// TwinCAT 3 PLC project plc_simple_move
// ProgramVersion: 3.1.0.8
// libraries:
//   Tc2_MC2, * (Beckhoff Automation GmbH)
//   Tc2_Standard, * (Beckhoff Automation GmbH)
//   Tc2_System, * (Beckhoff Automation GmbH)
//   Tc3_Interfaces, * (Beckhoff Automation GmbH)
//   Tc3_Module, * (Beckhoff Automation GmbH)
// project tree:
//   / PlcTask.TcTTO
//   POUs/ MAIN.TcPOU
// real-time tasks:
//   TASK PlcTask: cycle T#10ms, priority 20, ADS port 350
// motion (NC):
//   TASK NC-Task 1 SAF: cycle T#2ms, priority 4, ADS port 501
//   TASK NC-Task 1 SVB: cycle T#10ms, priority 8, ADS port 511
//   AXIS Axis 1 (id 1)
//     OtherSettings: AllowMotionCmdToSlave=true
//     encoder EncType=19
//       EncPara: MaxCount=#xffffffff
//     drive DrvType=16
//       DrvPara: MaxCount=#xffffffff
//         TimeComp: TaskDelayCycles=1
//     controller CtrType=1
//       CtrPara: PriorControlFactor=1
//         Observer: BandWidth=20
// I/O:
//   DEVICE Device 5 (EtherCAT), AmsNetId 5.39.221.128.6.1
//     Drive 12 (Elmo Drive) [Gold EtherCAT GCON Drive Rev:0x000103F6]
// variable links:
//   NC-Task 1 SAF/Axes/Axis 1 <-> Device 5 (EtherCAT)/Drive 12 (Elmo Drive)
//     Drive/Inputs/In/nDcOutputTime <-> InfoData/DcOutputShift
//     Drive/Inputs/In/nState1 <-> Inputs/Status word
//     Drive/Inputs/In/nState2 <-> Inputs/Status word @bit 8
//     Drive/Inputs/In/nState4 @bit 1 <-> WcState/InputToggle
//     Drive/Inputs/In/nState4 <-> WcState/WcState
//     Drive/Outputs/Out/nCtrl1 <-> Outputs/Control word
//     Drive/Outputs/Out/nCtrl2 <-> Outputs/Control word @bit 8
//     Drive/Outputs/Out/nDataOut1 <-> Outputs/Target Position
//     Enc/Inputs/In/nDataIn1 <-> Inputs/Position actual value
//     Enc/Inputs/In/nDcInputTime <-> InfoData/DcInputShift
//     Enc/Inputs/In/nState4 @bit 1 <-> WcState/InputToggle
//     Enc/Inputs/In/nState4 <-> WcState/WcState
//   plc_simple_move/plc_simple_move Instance <-> NC-Task 1 SAF/Axes/Axis 1
//     PlcTask Inputs/GVL.axis1.NcToPlc <-> Outputs/ToPlc
//     PlcTask Outputs/GVL.axis1.PlcToNc <-> Inputs/FromPlc

CONFIGURATION plc_simple_move
    RESOURCE PLC ON TwinCAT3
        TASK PlcTask(INTERVAL := T#10ms, PRIORITY := 20);
        PROGRAM MAIN WITH PlcTask : MAIN;
    END_RESOURCE
END_CONFIGURATION

// ---- POUs/MAIN.TcPOU
PROGRAM MAIN
VAR
	MC_Power_1: MC_Power;
	MC_MoveAbsolute_1: MC_MoveAbsolute;
	PowerEnable1: BOOL;				//供电使能
	MoveEnable1: BOOL;				//位移使能
	Pos1: LREAL;					//绝对位置
	Vel1: LREAL;					//速度
	PlcTime: LREAL := 0;			//PLC时间
	PlcCycleTicks: LREAL := 0.01;	//PLC运行循环时间 10ms
	tick: LREAL;					//计时开始时间
	WaitTime: LREAL;				//等待时间计时
	status: INT := 0;				//状态转移变量
	Move1Done: BOOL;
	axis1: AXIS_REF;
	star: BOOL := TRUE;
END_VAR

PlcTime := PlcTime + PlcCycleTicks;

MC_Power_1(
	Axis:= axis1, 
	Enable:= PowerEnable1, 
	Enable_Positive:= TRUE, 
	Enable_Negative:= TRUE, 
	Override:= , 
	BufferMode:= , 
	Options:= , 
	Status=> , 
	Busy=> , 
	Active=> , 
	Error=> , 
	ErrorID=> );
	
MC_MoveAbsolute_1(
	Axis:= axis1, 
	Execute:= MoveEnable1, 
	Position:= Pos1, 
	Velocity:= Vel1, 
	Acceleration:= , 
	Deceleration:= , 
	Jerk:= , 
	BufferMode:= , 
	Options:= , 
	Done=> Move1Done, 
	Busy=> , 
	Active=> , 
	CommandAborted=> , 
	Error=> , 
	ErrorID=> );


CASE status OF
	0://初始化
		PowerEnable1 := FALSE;
		MoveEnable1 := FALSE;
		status := 1;
		tick := PlcTime;	//为状态1计时设置启示时间
	1://等待3秒，供电&位移使能
		WaitTime := PlcTime-tick;
		IF WaitTime > 3 THEN
			PowerEnable1 := TRUE;
			status := 2;
			tick := PlcTime;	//为状态2计时设置启示时间
		END_IF
	2://设置移动距离&速度
		WaitTime := PlcTime-tick;
		IF WaitTime > 1 THEN
			Pos1 := 22;
			Vel1 := 1;
			MoveEnable1 := TRUE;
			status := 3;
		END_IF
	3://移动完成时停止
		IF Move1Done THEN
			status := 4;
		END_IF
	4://关闭
		MoveEnable1 := FALSE;
END_CASE

END_PROGRAM
